// TIA Portal V21 export
FUNCTION "GestScreensaver" : Void   // FC12, LAD
{ S7_Optimized_Access := 'TRUE' }
// stored: SetENOAutomatically false
   VAR_TEMP
      NumeroDiFrame : Int;
   END_VAR
BEGIN

REGION Network 1 (SCL)
   "T_ON"(I_CicloCPU := "CicloScansioneCPU_I".O_rCicloCpu,
          I_StartConteggio := NOT "Screensaver".DurataFrame.O,
          IO_DatiTimer := "Screensaver".DurataFrame);

   #NumeroDiFrame := 199;

   IF "Screensaver".TipoScreenSaver = 0 THEN
       IF "Screensaver".DurataFrame.O THEN
           IF NOT "Screensaver".DecrementaFrame THEN
               "Screensaver".Frameattuale += 1;
               IF "Screensaver".Frameattuale > #NumeroDiFrame THEN
                   "Screensaver".DecrementaFrame := True;
               END_IF;
           ELSE
               "Screensaver".Frameattuale -= 1;
               IF "Screensaver".Frameattuale <= 0 THEN
                   "Screensaver".DecrementaFrame := False;
               END_IF;
           END_IF;
       END_IF;
   END_IF;
END_REGION
END_FUNCTION
